FUNCTION_BLOCK newTaskGUIFB (* JADE WORKER *)
  (* Standard: 61499-1 *)
  (* Version 1.0, 2014-04-22, Ahmed, Fraunhofer IGD *)
  (* Compiler header: package fb.rt; *)
  (* Compiler Java Sun JDK 1.5.0 *)
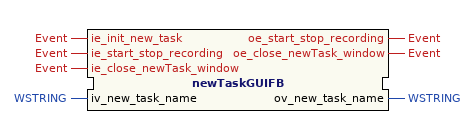
  EVENT_INPUT
    ie_init_new_task;
    ie_start_stop_recording;
    ie_close_newTask_window;
  END_EVENT
  EVENT_OUTPUT
    oe_start_stop_recording;
    oe_close_newTask_window;
  END_EVENT
  VAR_INPUT
    iv_new_task_name : WSTRING;
  END_VAR
  VAR_OUTPUT
    ov_new_task_name : WSTRING;
  END_VAR
END_FUNCTION_BLOCK
